FUNCTION_BLOCK SUB_2
  (* Standard: 61499-2 *)
  (* Version 10-09-13, slimrte *)
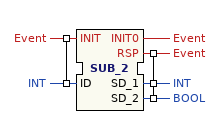
  EVENT_INPUT
    INIT WITH ID;
  END_EVENT
  EVENT_OUTPUT
    INIT0;
    RSP WITH SD_1, SD_2;
  END_EVENT
  VAR_INPUT
    ID : INT;
  END_VAR
  VAR_OUTPUT
    SD_1 : INT;
    SD_2 : BOOL;
  END_VAR
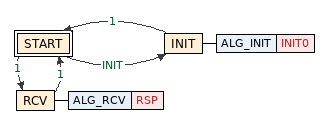
  EC_STATES
    START;
    RCV : ALG_RCV -> RSP;
    INIT : ALG_INIT -> INIT0;
  END_STATES
  EC_TRANSITIONS
    START TO INIT := INIT;
    INIT TO START := 1;
    START TO RCV := 1;
    RCV TO START := 1;
  END_TRANSITIONS
  ALGORITHM ALG_RCV IN Lua:
ASM       CONST 2  LOAD ID  NIRCV   IF GOTO process     GOTO out  process:    STORE SD_1    STORE SD_2  out:   END_ASM
  END_ALGORITHM
  ALGORITHM ALG_INIT IN Lua:

  END_ALGORITHM
END_FUNCTION_BLOCK
